// TwinCAT 3 PLC project Plc_IotMqttSampleIbmWatsonIot
// ProgramVersion: 3.1.4021.2
// libraries:
//   Tc2_Standard, * (Beckhoff Automation GmbH)
//   Tc2_System, * (Beckhoff Automation GmbH)
//   Tc2_Utilities, * (Beckhoff Automation GmbH)
//   Tc3_IotBase, * (Beckhoff Automation GmbH)
//   Tc3_Module, * (Beckhoff Automation GmbH)
// project tree:
//   / PlcTask.TcTTO
//   POUs/ MAIN.TcPOU, F_BuildJSON.TcPOU, PrgMqttCom.TcPOU
// real-time tasks:
//   TASK PlcTask: cycle T#10ms, priority 20, ADS port 350

CONFIGURATION Plc_IotMqttSampleIbmWatsonIot
    RESOURCE PLC ON TwinCAT3
        TASK PlcTask(INTERVAL := T#10ms, PRIORITY := 20);
        PROGRAM MAIN WITH PlcTask : MAIN;
    END_RESOURCE
END_CONFIGURATION

// ---- POUs/MAIN.TcPOU
PROGRAM MAIN
VAR
	m : INT;
END_VAR

m := m + 1;
PrgMqttCom();

END_PROGRAM

// ---- POUs/PrgMqttCom.TcPOU
PROGRAM PrgMqttCom
VAR
	fbMqttClient : FB_IotMqttClient;
	bSetParameter : BOOL := TRUE;
	bConnect : BOOL := TRUE;
	
	(* published message *)
	sTopicPub : STRING(255) := 'iot-2/evt/event_sensorData/fmt/json';
	{attribute 'TcEncoding':='UTF-8'}
	sPayloadPub : STRING(255);
	i: UDINT;
	fbTimer : TON := (PT:=T#500ms);
	fRandomSensor1 : LREAL;
	fRandomSensor2 : LREAL;
	fRandomSensor3 : LREAL;
	fbRandomNumber1 : DRAND;
	fbRandomNumber2 : DRAND;
	fbRandomNumber3 : DRAND;
		
	(* topic subscribtion *)
	bSubscribed : BOOL;
	sTopicSub : STRING(255) := 'iot-2/cmd/command_trigger/fmt/json';

	(* received message *)	
	{attribute 'TcEncoding':='UTF-8'}
	sTopicRcv : STRING(255);
	{attribute 'TcEncoding':='UTF-8'}
	sPayloadRcv : STRING(255);
	
	fbMessageQueue : FB_IotMqttMessageQueue;
	fbMessage : FB_IotMqttMessage;
		
	hrErrorOccurred : HRESULT; // contains the latest occurred error
END_VAR

IF bSetParameter THEN
	bSetParameter := FALSE;
	
	(* Broker settings für IBM Watson IoT *)
	fbMqttClient.sHostName := 'orgid.messaging.internetofthings.ibmcloud.com';
	fbMqttClient.nHostPort := 1883;
	fbMqttClient.sClientId := 'd:orgid:IPC:CX-12345'; 
	fbMqttClient.sUserName := 'use-token-auth';
	fbMqttClient.sUserPassword := '12342y?c12Gfq_8r12';
	
	fbMqttClient.ipMessageQueue := fbMessageQueue;
END_IF

fbMqttClient.Execute(bConnect);
IF fbMqttClient.bError THEN
	// add your error logging here
	hrErrorOccurred := fbMqttClient.hrErrorCode;
END_IF
IF fbMessageQueue.nQueuedMessages > 0 THEN
	IF fbMessageQueue.Dequeue(fbMessage:=fbMessage) THEN
		fbMessage.GetTopic(pTopic:=ADR(sTopicRcv), nTopicSize:=SIZEOF(sTopicRcv) );
		fbMessage.GetPayload(pPayload:=ADR(sPayloadRcv), nPayloadSize:=SIZEOF(sPayloadRcv), bSetNullTermination:=FALSE);
	END_IF
END_IF

IF fbMqttClient.bConnected THEN
	IF NOT bSubscribed THEN
		bSubscribed := fbMqttClient.Subscribe(sTopic:=sTopicSub, eQoS:=TcIotMqttQos.AtMostOnceDelivery);
		IF fbMqttClient.bError THEN
			// add your error logging here
			hrErrorOccurred := fbMqttClient.hrErrorCode;
		END_IF
	END_IF
	fbTimer(IN:=TRUE);
	IF fbTimer.Q THEN // publish new payload every second
		fbTimer(IN:=FALSE);
		i := i + 1;
		fbRandomNumber1(Seed:=1, Num=>fRandomSensor1);
		fbRandomNumber2(Seed:=2, Num=>fRandomSensor2);
		fbRandomNumber3(Seed:=3, Num=>fRandomSensor3);
		
		sPayloadPub := F_BuildJSON(	Sensor1 := LREAL_TO_STRING(fRandomSensor1*10), 
									Sensor2 := LREAL_TO_STRING(fRandomSensor2*10), 
									Sensor3 := LREAL_TO_STRING(fRandomSensor3*10)); 
		
		fbMqttClient.Publish(	sTopic:= sTopicPub, 
								pPayload:= ADR(sPayloadPub), nPayloadSize:= LEN2(ADR(sPayloadPub)), 
								eQoS:= TcIotMqttQos.AtMostOnceDelivery, bRetain:= FALSE, bQueue:= FALSE );
		IF fbMqttClient.bError THEN
			// add your error logging here
			hrErrorOccurred := fbMqttClient.hrErrorCode;
		END_IF
	END_IF
END_IF

END_PROGRAM

// ---- POUs/F_BuildJSON.TcPOU
FUNCTION F_BuildJSON : STRING(255)
VAR_INPUT
	  Sensor1 : STRING(255);
	  Sensor2 : STRING(255);
	  Sensor3 : STRING(255);
END_VAR
VAR
	  sReturnValue : STRING(255);
END_VAR

sReturnValue := CONCAT('{ "Sensor1" : ', Sensor1);
sReturnValue := CONCAT(sReturnValue, ', "Sensor2" : ');
sReturnValue := CONCAT(sReturnValue, Sensor2);
sReturnValue := CONCAT(sReturnValue, ', "Sensor3" : ');
sReturnValue := CONCAT(sReturnValue, Sensor3);
sReturnValue := CONCAT(sReturnValue, '}');
F_BuildJSON := sReturnValue;

END_FUNCTION
